// TIA Portal V21 export
ORGANIZATION_BLOCK "PidCyclicInterrupt"   // OB30, LAD, CyclicInterrupt
{ S7_Optimized_Access := 'TRUE' }
// stored: CyclicTime 50000, SetENOAutomatically false
BEGIN

REGION Network 1: "Fv1-Cv01" PID Block
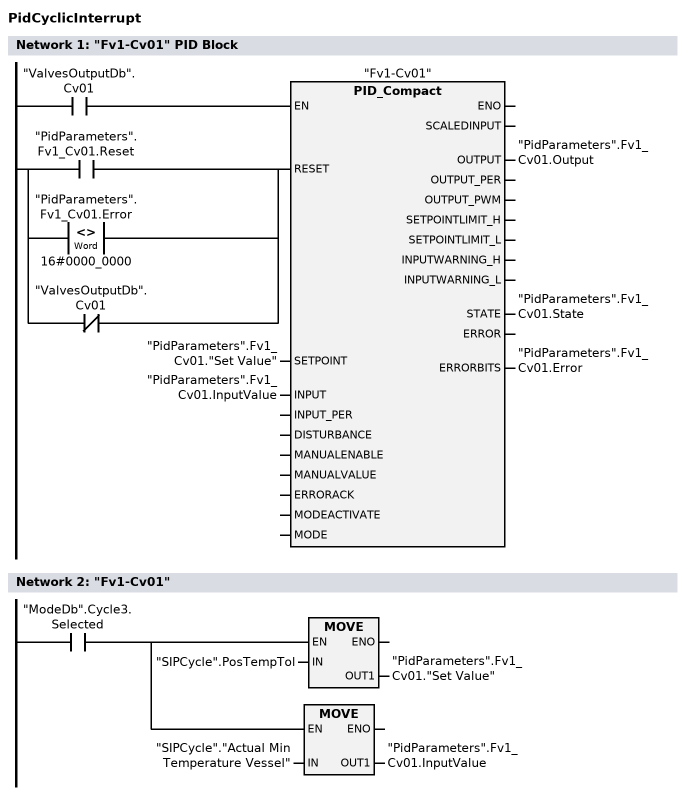
   RUNG wire#powerrail
      Contact( "ValvesOutputDb".Cv01 )
      "Fv1-Cv01".PID_Compact(Reset := wire#w1, Setpoint := "PidParameters".Fv1_Cv01."Set Value", Input := "PidParameters".Fv1_Cv01.InputValue, Input_PER :=, Disturbance :=, ManualEnable :=, ManualValue :=, ErrorAck :=, ModeActivate :=, Mode :=, ScaledInput =>, Output => "PidParameters".Fv1_Cv01.Output, Output_PER =>, Output_PWM =>, SetpointLimit_H =>, SetpointLimit_L =>, InputWarning_H =>, InputWarning_L =>, State => "PidParameters".Fv1_Cv01.State, Error =>, ErrorBits => "PidParameters".Fv1_Cv01.Error)
   END_RUNG
   RUNG wire#powerrail
      Contact( "PidParameters".Fv1_Cv01.Reset )
   END_RUNG wire#w1
   RUNG wire#powerrail
      { S7_Templates := "SrcType := Word" } NE_Contact(in1 := "PidParameters".Fv1_Cv01.Error, in2 := 16#0000_0000)
   END_RUNG wire#w1
   RUNG wire#powerrail
      I_Contact( "ValvesOutputDb".Cv01 )
   END_RUNG wire#w1
   // the same network as SCL:
   IF "ValvesOutputDb".Cv01 THEN
       "Fv1-Cv01"(Reset := "PidParameters".Fv1_Cv01.Reset OR ("PidParameters".Fv1_Cv01.Error <> 16#0000_0000) OR NOT "ValvesOutputDb".Cv01,   // PID_Compact
                  Setpoint := "PidParameters".Fv1_Cv01."Set Value",
                  Input := "PidParameters".Fv1_Cv01.InputValue,
                  Output => "PidParameters".Fv1_Cv01.Output,
                  State => "PidParameters".Fv1_Cv01.State,
                  ErrorBits => "PidParameters".Fv1_Cv01.Error);
   END_IF;
END_REGION

REGION Network 2: "Fv1-Cv01"
   RUNG wire#powerrail
      Contact( "ModeDb".Cycle3.Selected )
      wire#w1
      Move(in := "SIPCycle".PosTempTol, out1 => "PidParameters".Fv1_Cv01."Set Value")
   END_RUNG
   RUNG wire#w1
      Move(in := "SIPCycle"."Actual Min Temperature Vessel", out1 => "PidParameters".Fv1_Cv01.InputValue)
   END_RUNG
   // the same network as SCL:
   IF "ModeDb".Cycle3.Selected THEN
       "PidParameters".Fv1_Cv01."Set Value" := "SIPCycle".PosTempTol;
       "PidParameters".Fv1_Cv01.InputValue := "SIPCycle"."Actual Min Temperature Vessel";
   END_IF;
END_REGION
END_ORGANIZATION_BLOCK
